// TIA Portal V16 export
// export: Created 2023-03-29T11:05:04.4301754Z, ExportSetting WithDefaults, DisplayName Totally Integrated Automation Portal, DisplayVersion V16 Update 6, DisplayName TIA Portal Version Control Interface, DisplayVersion V16 Update 2, DisplayName TIA Portal Openness, DisplayVersion V16 Update 6, DisplayName STEP 7 Professional, DisplayVersion V16 Update 6, DisplayName STEP 7 Safety, DisplayVersion V16, DisplayName WinCC Advanced, DisplayVersion V16 Update 6
VAR_GLOBAL   // PLC tag table "ModbusRTU"
   setErrorModbsmasterFal AT %M18.0 : Bool;   // error bit modbus master falownik / Znacznik błedu komunikacji modbus
   setErrorModbsmasterMPP04_1 AT %M18.1 : Bool;   // error bit modbus master przepływomierz / Znacznik błedu komunikacji modbus
   setErrorModbsSlave AT %M18.2 : Bool;   // error bit modbus slave / Znacznik błedu komunikacji modbus
   "setErrorModbs----" AT %M18.3 : Bool;   // Znacznik błedu komunikacji modbus
   memRisErrorModbusmaster AT %M16.6 : Bool;   // Pamięć zbocza błędu komunikacji
   memReisModbus_Loop1 AT %M16.2 : Bool;   // Znacznik pamięci zbocza dla pętli 1
   memRisModbusmaster_Loop2 AT %M16.3 : Bool;   // pamięć zbocza dla petli 2 modbas
   memRisModbusmaster_Loop3 AT %M16.4 : Bool;   // pamięć zbocza pętli 3 modbas
   memRisModbus_Loop AT %M16.5 : Bool;   // Pamieć zbocza do uruchomienia petli SC1000
   ndrSlave AT %M16.7 : Bool;   // bit nowe dane gotowe / Pamieć zbocza błedu komunikacji
   drSlave AT %M14.5 : Bool;   // bit czytanie danych / pamięć zbocza błędu komunikacji
   memRisErrorModbusMPP04_1 AT %M14.6 : Bool;   // pamięć zbocza error modbus MPP04-1
   StatusSlave AT %MW29 : Word;   // Status slave Modbus RTU
   errorSatausSlave AT %MW31 : Word;   // Status błędu slave Modbus RTU
   setErrorModbsmasterMPP04_2 AT %M93.0 : Bool;   // error bit modbus master przepływomierz / Znacznik błedu komunikacji modbus
   memRisErrorModbusMPP04_2 AT %M14.7 : Bool;   // pamięć zbocza error modbus MPP04-1
   memRisErrorModbusFal AT %M93.1 : Bool;   // pamięć zbocza error modbus MPP04-1
   "memStep_errorMPP04-1" AT %MB100 : USInt;   // bajt pamieci w którym kroku nastąpił błąd modbus
   "memStep_errorMPP04-2" AT %MB101 : USInt;   // bajt pamieci w którym kroku nastąpił błąd modbus
   memStep_errorFal AT %MB102 : USInt;   // bajt pamieci w którym kroku nastąpił błąd modbus
   memStep_errorSlave AT %MB103 : USInt;   // bajt pamieci w którym kroku nastąpił błąd modbus
   "memRisSteperror_MPP04-1" AT %M104.0 : Bool;   // pamięć zbocza dla przechwycenia kroku błedu
   "memRisSteperror_MPP04-2" AT %M104.1 : Bool;   // pamięć zbocza dla przechwycenia kroku błedu
   memRisSteperror_Fal AT %M104.2 : Bool;   // pamięć zbocza dla przechwycenia kroku błedu
   memRisSteperror AT %M104.3 : Bool;   // pamięć zbocza dla przechwycenia kroku błedu
   act_flow_Q1 AT %MD600 : DWord;   // wartość przepływu Q1
   act_front_volumeVF_Q1 AT %MD604 : DWord;   // licznik objetości przód Q1
   act_back_valueVR_Q1 AT %MD608 : DWord;   // licznika objętości w tył Q1
   "act_differential counter VD_Q1" AT %MD612 : DWord;   // liczni różnicowyobjętości VD Q1
   "act_volume counter status _GF_Q1" AT %MD616 : DWord;   // główny licznik objetosci przód GF Q1
   "act_volume counter status_GR_Q1" AT %MD620 : DWord;   // główny licznik objetości w tył GR Q1
   "act_differential counter status_GD_Q1" AT %MD624 : DWord;   // główny różnicow licznik objetości GD Q1
   act_flow_Q2 AT %MD630 : DWord;   // wartość przepływu Q2
   act_ValueVF_Q2 AT %MD634 : DWord;   // licznik objetości przód Q2
   act_front_volumeVF_Q2 AT %MD638 : DWord;   // licznika objętości w tył Q2
   act_back_balueVR_Q2 AT %MD642 : DWord;   // liczni różnicowyobjętości VD Q2
   "act_differential counter VD_Q2" AT %MD646 : DWord;   // główny licznik objetosci przód GF Q2
   "act_volume counter status _GF_Q2" AT %MD650 : DWord;   // główny licznik objetości w tył GR Q2
   "act_volume counter status_GR_Q2" AT %MD654 : DWord;   // główny różnicow licznik objetości GD Q2
   "act_differential counter status_GD_Q2" AT %MD658 : DWord;
   Switch_PrzepłtwSygnał AT %M92.0 : Bool;   // wybór źródła wartości pomiaru analog / modbus rtu
END_VAR
